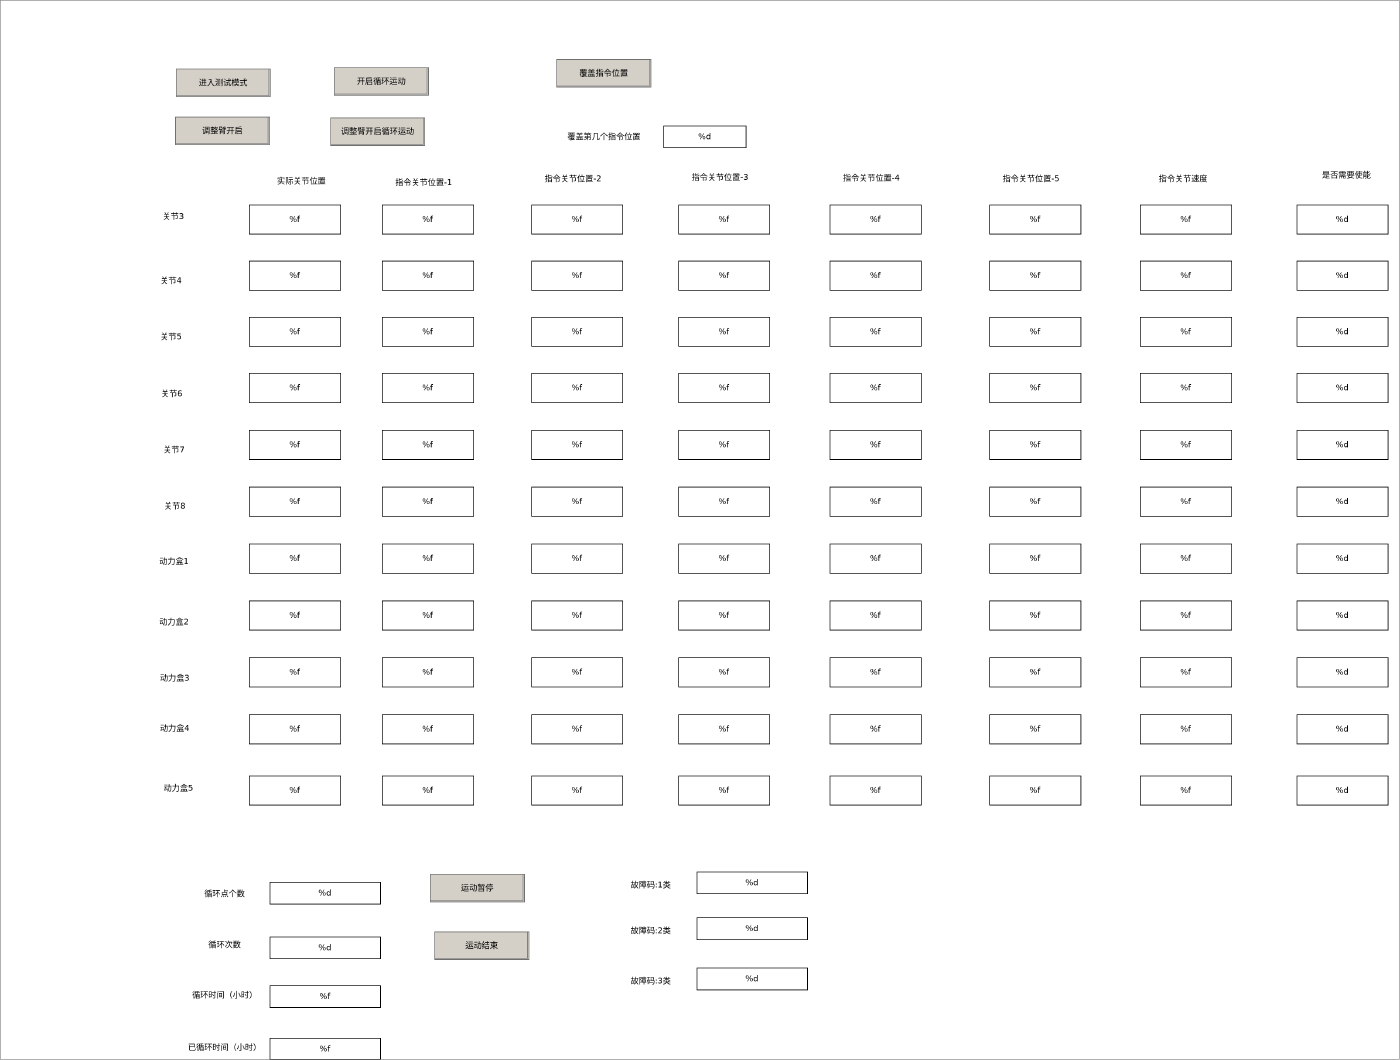
VISUALIZATION cycle_a2  // 1895x1435
    Button (238,93 128x38), "进入测试模式", colour toggle: g_cycleTest.m_enterCycleTestMode[2]
        toggle g_cycleTest.m_enterCycleTestMode[2]
    Button (452,91 128x38), "开启循环运动", colour toggle: g_cycleTest.m_startMotion[2]
        toggle g_cycleTest.m_startMotion[2]
    Label (501,233 145x28), "指令关节位置-1"
    Label (333,230 150x30), "实际关节位置"
    Rectangle (337,505 124x40), "%f", text variable: g_cycleTest.m_actJntPos[2][1]
    Label (162,279 145x28), "关节3"
    Label (159,366 145x28), "关节4"
    Label (159,442 145x28), "关节5"
    Label (160,519 145x28), "关节6"
    Label (163,595 145x28), "关节7"
    Label (164,671 145x28), "关节8"
    Label (163,746 145x28), "动力盒1"
    Label (163,828 145x28), "动力盒2"
    Label (169,1053 145x28), "动力盒5"
    Label (164,904 145x28), "动力盒3"
    Label (164,972 145x28), "动力盒4"
    Rectangle (337,582 124x40), "%f", text variable: g_cycleTest.m_actJntPos[2][2]
    Rectangle (337,659 124x40), "%f", text variable: g_cycleTest.m_actJntPos[2][3]
    Rectangle (337,736 124x40), "%f", text variable: g_cycleTest.m_actJntPos[2][4]
    Rectangle (337,813 124x40), "%f", text variable: g_cycleTest.m_actJntPos[2][5]
    Rectangle (337,890 124x40), "%f", text variable: g_cycleTest.m_actJntPos[2][6]
    Rectangle (337,967 124x40), "%f", text variable: g_cycleTest.m_actJntPos[2][7]
    Rectangle (337,1050 124x40), "%f", text variable: g_cycleTest.m_actJntPos[2][8]
    Rectangle (337,277 124x40), "%f", text variable: g_cycleTest.m_actJntPosSetup[2][3]
    Rectangle (337,353 124x40), "%f", text variable: g_cycleTest.m_actJntPosSetup[2][4]
    Rectangle (337,429 124x40), "%f", text variable: g_cycleTest.m_actJntPosSetup[2][5]
    Rectangle (517,277 124x40), "%f", text variable: g_cycleTest.m_targetJntPosSetup[2,1][3]
        OnMouseClick: write the text variable via Default
    Rectangle (517,353 124x40), "%f", text variable: g_cycleTest.m_targetJntPosSetup[2,1][4]
        OnMouseClick: write the text variable via Default
    Rectangle (517,429 124x40), "%f", text variable: g_cycleTest.m_targetJntPosSetup[2,1][5]
        OnMouseClick: write the text variable via Default
    Rectangle (517,505 124x40), "%f", text variable: g_cycleTest.m_targetJntPos[2,1][1]
        OnMouseClick: write the text variable via Default
    Rectangle (517,582 124x40), "%f", text variable: g_cycleTest.m_targetJntPos[2,1][2]
        OnMouseClick: write the text variable via Default
    Rectangle (517,659 124x40), "%f", text variable: g_cycleTest.m_targetJntPos[2,1][3]
        OnMouseClick: write the text variable via Default
    Rectangle (517,736 124x40), "%f", text variable: g_cycleTest.m_targetJntPos[2,1][4]
        OnMouseClick: write the text variable via Default
    Rectangle (517,813 124x40), "%f", text variable: g_cycleTest.m_targetJntPos[2,1][5]
        OnMouseClick: write the text variable via Default
    Rectangle (517,890 124x40), "%f", text variable: g_cycleTest.m_targetJntPos[2,1][6]
        OnMouseClick: write the text variable via Default
    Rectangle (517,967 124x40), "%f", text variable: g_cycleTest.m_targetJntPos[2,1][7]
        OnMouseClick: write the text variable via Default
    Rectangle (517,1050 124x40), "%f", text variable: g_cycleTest.m_targetJntPos[2,1][8]
        OnMouseClick: write the text variable via Default
    Label (703,228 145x28), "指令关节位置-2"
    Rectangle (719,277 124x40), "%f", text variable: g_cycleTest.m_targetJntPosSetup[2,2][3]
        OnMouseClick: write the text variable via Default
    Rectangle (719,353 124x40), "%f", text variable: g_cycleTest.m_targetJntPosSetup[2,2][4]
        OnMouseClick: write the text variable via Default
    Rectangle (719,429 124x40), "%f", text variable: g_cycleTest.m_targetJntPosSetup[2,2][5]
        OnMouseClick: write the text variable via Default
    Rectangle (719,505 124x40), "%f", text variable: g_cycleTest.m_targetJntPos[2,2][1]
        OnMouseClick: write the text variable via Default
    Rectangle (719,582 124x40), "%f", text variable: g_cycleTest.m_targetJntPos[2,2][2]
        OnMouseClick: write the text variable via Default
    Rectangle (719,659 124x40), "%f", text variable: g_cycleTest.m_targetJntPos[2,2][3]
        OnMouseClick: write the text variable via Default
    Rectangle (719,736 124x40), "%f", text variable: g_cycleTest.m_targetJntPos[2,2][4]
        OnMouseClick: write the text variable via Default
    Rectangle (719,813 124x40), "%f", text variable: g_cycleTest.m_targetJntPos[2,2][5]
        OnMouseClick: write the text variable via Default
    Rectangle (719,890 124x40), "%f", text variable: g_cycleTest.m_targetJntPos[2,2][6]
        OnMouseClick: write the text variable via Default
    Rectangle (719,967 124x40), "%f", text variable: g_cycleTest.m_targetJntPos[2,2][7]
        OnMouseClick: write the text variable via Default
    Rectangle (719,1050 124x40), "%f", text variable: g_cycleTest.m_targetJntPos[2,2][8]
        OnMouseClick: write the text variable via Default
    Label (902,226 145x28), "指令关节位置-3"
    Rectangle (918,277 124x40), "%f", text variable: g_cycleTest.m_targetJntPosSetup[2,3][3]
        OnMouseClick: write the text variable via Default
    Rectangle (918,353 124x40), "%f", text variable: g_cycleTest.m_targetJntPosSetup[2,3][4]
        OnMouseClick: write the text variable via Default
    Rectangle (918,429 124x40), "%f", text variable: g_cycleTest.m_targetJntPosSetup[2,3][5]
        OnMouseClick: write the text variable via Default
    Rectangle (918,505 124x40), "%f", text variable: g_cycleTest.m_targetJntPos[2,3][1]
        OnMouseClick: write the text variable via Default
    Rectangle (918,582 124x40), "%f", text variable: g_cycleTest.m_targetJntPos[2,3][2]
        OnMouseClick: write the text variable via Default
    Rectangle (918,659 124x40), "%f", text variable: g_cycleTest.m_targetJntPos[2,3][3]
        OnMouseClick: write the text variable via Default
    Rectangle (918,736 124x40), "%f", text variable: g_cycleTest.m_targetJntPos[2,3][4]
        OnMouseClick: write the text variable via Default
    Rectangle (918,813 124x40), "%f", text variable: g_cycleTest.m_targetJntPos[2,3][5]
        OnMouseClick: write the text variable via Default
    Rectangle (918,890 124x40), "%f", text variable: g_cycleTest.m_targetJntPos[2,3][6]
        OnMouseClick: write the text variable via Default
    Rectangle (918,967 124x40), "%f", text variable: g_cycleTest.m_targetJntPos[2,3][7]
        OnMouseClick: write the text variable via Default
    Rectangle (918,1050 124x40), "%f", text variable: g_cycleTest.m_targetJntPos[2,3][8]
        OnMouseClick: write the text variable via Default
    Label (1107,227 145x28), "指令关节位置-4"
    Rectangle (1123,277 124x40), "%f", text variable: g_cycleTest.m_targetJntPosSetup[2,4][3]
        OnMouseClick: write the text variable via Default
    Rectangle (1123,353 124x40), "%f", text variable: g_cycleTest.m_targetJntPosSetup[2,4][4]
        OnMouseClick: write the text variable via Default
    Rectangle (1123,429 124x40), "%f", text variable: g_cycleTest.m_targetJntPosSetup[2,4][5]
        OnMouseClick: write the text variable via Default
    Rectangle (1123,505 124x40), "%f", text variable: g_cycleTest.m_targetJntPos[2,4][1]
        OnMouseClick: write the text variable via Default
    Rectangle (1123,582 124x40), "%f", text variable: g_cycleTest.m_targetJntPos[2,4][2]
        OnMouseClick: write the text variable via Default
    Rectangle (1123,659 124x40), "%f", text variable: g_cycleTest.m_targetJntPos[2,4][3]
        OnMouseClick: write the text variable via Default
    Rectangle (1123,736 124x40), "%f", text variable: g_cycleTest.m_targetJntPos[2,4][4]
        OnMouseClick: write the text variable via Default
    Rectangle (1123,813 124x40), "%f", text variable: g_cycleTest.m_targetJntPos[2,4][5]
        OnMouseClick: write the text variable via Default
    Rectangle (1123,890 124x40), "%f", text variable: g_cycleTest.m_targetJntPos[2,4][6]
        OnMouseClick: write the text variable via Default
    Rectangle (1123,967 124x40), "%f", text variable: g_cycleTest.m_targetJntPos[2,4][7]
        OnMouseClick: write the text variable via Default
    Rectangle (1123,1050 124x40), "%f", text variable: g_cycleTest.m_targetJntPos[2,4][8]
        OnMouseClick: write the text variable via Default
    Label (1323,228 145x28), "指令关节位置-5"
    Rectangle (1339,277 124x40), "%f", text variable: g_cycleTest.m_targetJntPosSetup[2,5][3]
        OnMouseClick: write the text variable via Default
    Rectangle (1339,353 124x40), "%f", text variable: g_cycleTest.m_targetJntPosSetup[2,5][4]
        OnMouseClick: write the text variable via Default
    Rectangle (1339,429 124x40), "%f", text variable: g_cycleTest.m_targetJntPosSetup[2,5][5]
        OnMouseClick: write the text variable via Default
    Rectangle (1339,505 124x40), "%f", text variable: g_cycleTest.m_targetJntPos[2,5][1]
        OnMouseClick: write the text variable via Default
    Rectangle (1339,582 124x40), "%f", text variable: g_cycleTest.m_targetJntPos[2,5][2]
        OnMouseClick: write the text variable via Default
    Rectangle (1339,659 124x40), "%f", text variable: g_cycleTest.m_targetJntPos[2,5][3]
        OnMouseClick: write the text variable via Default
    Rectangle (1339,736 124x40), "%f", text variable: g_cycleTest.m_targetJntPos[2,5][4]
        OnMouseClick: write the text variable via Default
    Rectangle (1339,813 124x40), "%f", text variable: g_cycleTest.m_targetJntPos[2,5][5]
        OnMouseClick: write the text variable via Default
    Rectangle (1339,890 124x40), "%f", text variable: g_cycleTest.m_targetJntPos[2,5][6]
        OnMouseClick: write the text variable via Default
    Rectangle (1339,967 124x40), "%f", text variable: g_cycleTest.m_targetJntPos[2,5][7]
        OnMouseClick: write the text variable via Default
    Rectangle (1339,1050 124x40), "%f", text variable: g_cycleTest.m_targetJntPos[2,5][8]
        OnMouseClick: write the text variable via Default
    Button (237,158 128x38), "调整臂开启", colour toggle: g_cycleTest.m_enterCycleTestModeSetup[2]
        toggle g_cycleTest.m_enterCycleTestModeSetup[2]
    Button (447,159 128x38), "调整臂开启循环运动", colour toggle: g_cycleTest.m_startMotionSetup[2]
        toggle g_cycleTest.m_startMotionSetup[2]
    Label (1529,228 145x28), "指令关节速度"
    Rectangle (1543,277 124x40), "%f", text variable: g_cycleTest.m_targetJntVelSetup[2][3]
        OnMouseClick: write the text variable via Default
    Rectangle (1543,353 124x40), "%f", text variable: g_cycleTest.m_targetJntVelSetup[2][4]
        OnMouseClick: write the text variable via Default
    Rectangle (1543,429 124x40), "%f", text variable: g_cycleTest.m_targetJntVelSetup[2][5]
        OnMouseClick: write the text variable via Default
    Rectangle (1543,505 124x40), "%f", text variable: g_cycleTest.m_targetJntVelN8[2][1]
        OnMouseClick: write the text variable via Default
    Rectangle (1543,582 124x40), "%f", text variable: g_cycleTest.m_targetJntVelN8[2][2]
        OnMouseClick: write the text variable via Default
    Rectangle (1543,659 124x40), "%f", text variable: g_cycleTest.m_targetJntVelN8[2][3]
        OnMouseClick: write the text variable via Default
    Rectangle (1543,736 124x40), "%f", text variable: g_cycleTest.m_targetJntVelN8[2][4]
        OnMouseClick: write the text variable via Default
    Rectangle (1543,813 124x40), "%f", text variable: g_cycleTest.m_targetJntVelN8[2][5]
        OnMouseClick: write the text variable via Default
    Rectangle (1543,890 124x40), "%f", text variable: g_cycleTest.m_targetJntVelN8[2][6]
        OnMouseClick: write the text variable via Default
    Rectangle (1543,967 124x40), "%f", text variable: g_cycleTest.m_targetJntVelN8[2][7]
        OnMouseClick: write the text variable via Default
    Rectangle (1543,1050 124x40), "%f", text variable: g_cycleTest.m_targetJntVelN8[2][8]
        OnMouseClick: write the text variable via Default
    Label (229,1195 150x30), "循环点个数"
    Rectangle (365,1194 150x30), "%d", text variable: g_cycleTest.m_pointSum[2]
        OnMouseClick: write the text variable via Default
    Rectangle (365,1268 150x30), "%d", text variable: g_cycleTest.m_curCycleNum[2]
        OnMouseClick: write the text variable via Default
    Label (229,1264 150x30), "循环次数"
    Button (582,1183 128x38), "运动暂停", colour toggle: g_cycleTest.m_pause[2]
        toggle g_cycleTest.m_pause[2]
    Button (588,1261 128x38), "运动结束", colour toggle: g_cycleTest.m_finish[2]
        tap g_cycleTest.m_finish[2]
    Rectangle (365,1334 150x30), "%f", text variable: g_cycleTest.m_tgtCycleTime[2]
        OnMouseClick: write the text variable via Default
    Label (229,1332 150x30), "循环时间（小时）"
    Rectangle (365,1405 150x30), "%f", text variable: g_cycleTest.m_curCycleTime[2]
        OnMouseClick: write the text variable via Default
    Label (229,1403 150x30), "已循环时间（小时）"
    Button (753,80 128x38), "覆盖指令位置", colour toggle: g_cycleTest.m_coverCmdPos[2]
        tap g_cycleTest.m_coverCmdPos[2]
    Rectangle (898,170 112x30), "%d", text variable: g_cycleTest.m_pntIdForCoverCmd[2]
        OnMouseClick: write the text variable via Default
    Label (745,171 145x28), "覆盖第几个指令位置"
    Label (1750,222 145x30), "是否需要使能"
    Rectangle (1755,277 124x40), "%d", text variable: g_cycleTest.m_jntEnableSetup[2][3]
        OnMouseClick: write the text variable via Default
    Rectangle (1755,353 124x40), "%d", text variable: g_cycleTest.m_jntEnableSetup[2][4]
        OnMouseClick: write the text variable via Default
    Rectangle (1755,429 124x40), "%d", text variable: g_cycleTest.m_jntEnableSetup[2][5]
        OnMouseClick: write the text variable via Default
    Rectangle (1755,505 124x40), "%d", text variable: g_cycleTest.m_jntEnable[2][1]
        OnMouseClick: write the text variable via Default
    Rectangle (1755,582 124x40), "%d", text variable: g_cycleTest.m_jntEnable[2][2]
        OnMouseClick: write the text variable via Default
    Rectangle (1755,659 124x40), "%d", text variable: g_cycleTest.m_jntEnable[2][3]
        OnMouseClick: write the text variable via Default
    Rectangle (1755,736 124x40), "%d", text variable: g_cycleTest.m_jntEnable[2][4]
        OnMouseClick: write the text variable via Default
    Rectangle (1755,813 124x40), "%d", text variable: g_cycleTest.m_jntEnable[2][5]
        OnMouseClick: write the text variable via Default
    Rectangle (1755,890 124x40), "%d", text variable: g_cycleTest.m_jntEnable[2][6]
        OnMouseClick: write the text variable via Default
    Rectangle (1755,967 124x40), "%d", text variable: g_cycleTest.m_jntEnable[2][7]
        OnMouseClick: write the text variable via Default
    Rectangle (1755,1050 124x40), "%d", text variable: g_cycleTest.m_jntEnable[2][8]
        OnMouseClick: write the text variable via Default
    Rectangle (943,1180 150x30), "%d", text variable: GVL_interactUI.g_errIdType1
        OnMouseClick: write the text variable via Default
    Label (806,1183 150x30), "故障码:1类"
    Rectangle (943,1242 150x30), "%d", text variable: GVL_interactUI.g_errIdType2
        OnMouseClick: write the text variable via Default
    Label (806,1245 150x30), "故障码:2类"
    Rectangle (943,1310 150x30), "%d", text variable: GVL_interactUI.g_errIdType3
        OnMouseClick: write the text variable via Default
    Label (806,1313 150x30), "故障码:3类"
END_VISUALIZATION

(* stored: Version 1.1.0.1, ProductVersion 3.1.4024.11
   Visu cycle_a2: Id {28a6998e-2011-4836-9c53-d1152735d421} *)
